{attribute 'OPC.UA.DA.StructuredType' := '1'}
FUNCTION_BLOCK FB_DosingPumpAgrowtek_R2_Batch EXTENDS FB_BaseDevice IMPLEMENTS I_PumpDosing

VAR_IN_OUT
	{attribute 'OPC.UA.DA' := '0'}
	//fbModbusMaster: FB_ModbusMaster;
	fbModbusManager: FB_ModbusManager;
	
	bInitialDose: BOOL := FALSE; // this is set to TRUE when the nDoseQTYMls is pre-loaded for the initial dose sequence. Setting nDoseQtyML or executing doses from control loops is disabled when this is true
END_VAR

VAR_INPUT
	nModbusUnitID: UINT; 
END_VAR

VAR
	// Modbus Variables
	nPumpID: UINT;	// Pump ID is different to the modbus ID because there are 5 pumps on the 1 modbus address
	 
	ePumpType: E_DosingPump;

	
	bEnableComms: BOOL := TRUE;
	bFirtRun: BOOL := TRUE;
	bResetTimer: BOOL := TRUE;
	
	// Async Statemachine Variables
	{attribute 'OPC.UA.DA' := '0'}
	eSMState: (WAIT, SET_TIME, GET_TIME, SET_SPEED, FINISH);
	
	// Dosing Variables
	{attribute 'OPC.UA.DA' := '0'} 
	fbTONdoseTime: TON;  
	{attribute 'OPC.UA.DA' := '1'} 
	nDoseRateMLph: UINT;
	{attribute 'OPC.UA.DA' := '1'} 
	nDoseQtyMls: REAL;
	{attribute 'OPC.UA.DA' := '1'} 
	tTimeToDose: TIME;
	
	nTimeToDoseSeconds: INT;
	nRetries: INT := 0;
	
	// delay between writing pump speed and reading pump speed
	fbTON_WaitForMsg : TON := (PT := T#1S);

	// Variables updated over Modbus
	{attribute 'OPC.UA.DA' := '1'} 
	nPumpSpeed_Requested: UINT;
	
	{attribute 'OPC.UA.DA' := '1'} 
	nPumpSpeed: UINT;
	{attribute 'OPC.UA.DA' := '1'} 
	nPumpRunTime: UINT; 
	
	
	
	
	bDoseRequestSent:		BOOL := FALSE;
	bDoseRequestComplete: 	BOOL := FALSE;
	
	tDataRefresh: TIME := T#10S;
	fbTON_DataRefresh: 	TON := (PT := tDataRefresh, IN := FALSE);
	fbTON_MsgTimeout: 	TON := (PT := T#4S, IN := FALSE);
	
	// Modbus Requests
	stModRead_MotorSpeed: 	ST_Modbus_ReadRequest;
	stModRead_MotorRunTime: ST_Modbus_ReadRequest;
	stModWrite_MotorSpeed: 	ST_Modbus_WriteRequest;
	stModWrite_SetID: 		ST_Modbus_WriteRequest;
	stModWrite_Timeout:	ST_Modbus_WriteRequest;
	stModRead_Timeout:	ST_Modbus_ReadRequest;
	
	
	bRaiseError1: BOOL := FALSE;
	bClearError: BOOL := FALSE;
	bRaiseError2: BOOL := FALSE;
	
	
END_VAR

fbTONdoseTime();
fbTON_MsgTimeout();
fbTON_DataRefresh();
fbTON_WaitForMsg();

IF GVL.bAutoUpdateDeviceState THEN
	eState := eStateTarget;	
END_IF

IF (eStateTarget = E_DeviceState.RUNNING) AND (eState := E_DeviceState.IDLE) THEN  // this is used to handle the initial batch dose commands from the sequene manager (this control loop uses the executeDOse method
	executeDose(DoseQtyMls := nDoseQtyMls, DoseRateMlph := 40, RequestComplete := ADR(bDoseRequestSent));
	eState := E_DeviceState.RUNNING;
END_IF


IF bFirtRun THEN
	init_ModbusRequests();
	bFirtRun := FALSE;
END_IF

IF eMode = E_DeviceMode.MANUAL THEN
	bEnable := TRUE;
END_IF


IF bResetTimer THEN
	fbTON_DataRefresh.IN := TRUE;
	bResetTimer := FALSE;
END_IF

// Asynchronous update of local variables from the Modbus request structures
nPumpSpeed 		:= WORD_TO_UINT(stModRead_MotorSpeed.ReadRegsVals[1]);
nPumpRunTime 	:= WORD_TO_UINT(stModRead_MotorRunTime.ReadRegsVals[1]);
	

CASE eSMState OF

	WAIT:
		eState := E_DeviceState.IDLE;
		fbTON_WaitForMsg(IN := FALSE);
		
	SET_TIME:
		eState := E_DeviceState.RUNNING;
		stModWrite_Timeout.WriteRegVals[1] := INT_TO_WORD(nTimeToDoseSeconds);
		fbModbusManager.addRequest_Write_Priority(WriteRequest := ADR(stModWrite_Timeout));
		fbTON_WaitForMsg(IN := TRUE);
		eSMState := GET_TIME;
		
		
	GET_TIME:
		IF stModRead_Timeout.ReadRegsVals[1] = INT_TO_WORD(nTimeToDoseSeconds) THEN
			stModRead_Timeout.ReadRegsVals[1] := 0;
			fbTON_WaitForMsg(IN := FALSE);
			eSMState := SET_SPEED;
		ELSE
			fbTON_WaitForMsg(IN := TRUE);
		END_IF
	
		IF fbTON_WaitForMsg.Q THEN
			fbModbusManager.addRequest_Read_Priority(ReadRequest := ADR(stModRead_Timeout));	
			fbTON_WaitForMsg(IN := FALSE);
		ELSE
			fbTON_WaitForMsg(IN := FALSE);			// add retry counter here
			nRetries := nRetries + 1;
			IF nRetries > 5 THEN
				eSMState := WAIT;
				eState := E_DeviceState.IDLE;
				bBusy := FALSE;
				nRetries := 0;
				raiseAlarm(Priority := E_AlarmPriority.High, Label := 'Motor Failed to Receive Duration Command After 5 Retries', Enabled := TRUE, DeviceAlarmID := 1);
			END_IF
		END_IF
		
	SET_SPEED:
		fbTON_WaitForMsg(IN := TRUE);
		
		IF fbTON_WaitForMsg.Q THEN
			stModWrite_MotorSpeed.WriteRegVals[1] := UINT_TO_WORD(nPumpSpeed_Requested);
			fbModbusManager.addRequest_Write_Priority(WriteRequest := stModWrite_MotorSpeed);
			fbTON_WaitForMsg(IN := FALSE);
			eSMState := FINISH;
		END_IF
		
	FINISH:
		fbTON_WaitForMsg(IN := TRUE);
		
		IF fbTON_WaitForMsg.Q THEN
			fbModbusManager.addRequest_Read_Priority(ReadRequest := ADR(stModRead_Timeout));	
			fbTON_WaitForMsg(IN := FALSE);
		END_IF
		
		IF stModRead_Timeout.ReadRegsVals[1] = 0 THEN
			eSMState := WAIT;
			bBusy := FALSE;
			eState := E_DeviceState.IDLE;
			bInitialDose := FALSE;
		ELSE
			nRetries := nRetries + 1;
			IF nRetries > 5 THEN
				raiseAlarm(Priority := E_AlarmPriority.High, Label := 'Motor Counter Failed to Reach 0 After 5 Retries', Enabled := TRUE, DeviceAlarmID := 2);
				nRetries := 0;
				bBusy := FALSE;
				eSMState := WAIT;
				eState := E_DeviceState.IDLE;
				bInitialDose := FALSE;	
			END_IF
		END_IF

END_CASE

{warning 'add method implementation '}
METHOD executeDose : BOOL
VAR_INPUT
	DoseQtyMls: LREAL;
	DoseRateMlph: UINT;
	RequestComplete: 	POINTER TO BOOL;
END_VAR
VAR_OUTPUT
	RequestAccepted: BOOL;
END_VAR
(* setDose dispenses the amount requested at a user requested dose rate *)

IF ((bEnable AND bEnableComms) OR (eMode = E_DeviceMode.MANUAL)) AND ( NOT bInitialDose)  THEN
	
		nPumpSpeed_Requested := 40;
		tTimeToDose := REAL_TO_TIME(( ABS(DoseQtyMls) / (480.0*(UINT_TO_REAL(nPumpSpeed_Requested)/100.0))) * 60.0 *1000.0);  // Agrowtek maximum flow rate is 480 ml/min
		fbTONdoseTime.PT := tTimeToDose;
	
		IF tTimeToDose >= T#1S THEN
			nTimeToDoseSeconds := (TIME_TO_INT(tTimeToDose)/1000);
			nDoseQtyMls := nTimeToDoseSeconds * ((nPumpSpeed_Requested/100.0) * (480.0/60.0));
			eSMState := SET_TIME;
			eState := E_Devicestate.RUNNING;
			bBusy := TRUE;	
		END_IF
	END_IF
END_METHOD

METHOD FB_init : BOOL


VAR_INPUT
	bInitRetains : BOOL; // if TRUE, the retain variables are initialized (warm start / cold start)
	bInCopyCode : BOOL;  // if TRUE, the instance afterwards gets moved into the copy code (online change)
	
	PumpID: STRING;
	PumpDescription: STRING;
	PumpType: E_DosingPump;
	ManifoldModbusID: UINT; 
	
END_VAR
sID := PumpID;
sDescr := PumpDescription;
ePumpType := PumpType;
nModbusUnitID := ManifoldModbusID;
END_METHOD

METHOD getAdrMotorTime : UINT
VAR_INPUT
	PumpType: E_DosingPump;
END_VAR
// This method retrieves the Modbus register for the individual Agrowtek pump
// We need to do this because 5 pumps share the same Modbus slave ID, however have differing registers to write to

CASE PumpType OF
	
	E_DosingPump.PH_DOWN:
		getAdrReadWriteSpeed := 200;
		
	E_DosingPump.NUTRIENT_A:
		getAdrReadWriteSpeed := 201;
		
	E_DosingPump.NUTRIENT_B:
		getAdrReadWriteSpeed := 202;
		
	E_DosingPump.NUTRIENT_C:
		getAdrReadWriteSpeed := 203;
		
	E_DosingPump.PH_UP:
		getAdrReadWriteSpeed := 204;
		
END_CASE
END_METHOD

METHOD getAdrReadAccumRunTime : UINT
VAR_INPUT
	PumpType: E_DosingPump;
END_VAR

VAR
	Address: UINT;
END_VAR
// This method retrieves the Modbus register for the individual Agrowtek pump
// We need to do this because 5 pumps share the same Modbus slave ID, however have differing registers to write to

CASE PumpType OF
	
	E_DosingPump.PH_DOWN:
		Address := 16#64;
		
	E_DosingPump.NUTRIENT_A:
		Address := 16#65;
		
	E_DosingPump.NUTRIENT_B:
		Address := 16#66;

	E_DosingPump.NUTRIENT_C:
		Address := 16#67;
		
	E_DosingPump.PH_UP:
		Address := 16#68;
		
END_CASE

getAdrReadAccumRunTime := Address;
END_METHOD

METHOD getAdrReadWriteSpeed : UINT
VAR_INPUT
	PumpType: E_DosingPump;
END_VAR
// This method retrieves the Modbus register for the individual Agrowtek pump
// We need to do this because 5 pumps share the same Modbus slave ID, however have differing registers to write to

CASE PumpType OF
	
	E_DosingPump.PH_DOWN:
		getAdrReadWriteSpeed := 16#64;
		
	E_DosingPump.NUTRIENT_A:
		getAdrReadWriteSpeed := 16#65;
		
	E_DosingPump.NUTRIENT_B:
		getAdrReadWriteSpeed := 16#66;
		
	E_DosingPump.NUTRIENT_C:
		getAdrReadWriteSpeed := 16#67;
		
	E_DosingPump.PH_UP:
		getAdrReadWriteSpeed := 16#68;
		
END_CASE
END_METHOD

METHOD init_ModbusRequests : BOOL
VAR_INPUT
END_VAR
stModRead_MotorSpeed.SlaveAddress := nModbusUnitID;			
stModRead_MotorSpeed.AdrFirstSlaveRegisterRead := getAdrReadWriteSpeed(PumpType := ePumpType);
stModRead_MotorSpeed.QtyWordsToRead := 1;				// The value is a 16-bit word
stModRead_MotorSpeed.bRequestAccepted := FALSE;
stModRead_MotorSpeed.bRequestCompleted := FALSE;
stModRead_MotorSpeed.ReadRegsVals := GVL.ModbusEmptyBuffer;

stModRead_MotorRunTime.SlaveAddress := nModbusUnitID;			
stModRead_MotorRunTime.AdrFirstSlaveRegisterRead := getAdrReadAccumRunTime(PumpType := ePumpType);
stModRead_MotorRunTime.QtyWordsToRead := 1;				// The value is a 32-bit word
stModRead_MotorRunTime.bRequestAccepted := FALSE;
stModRead_MotorRunTime.bRequestCompleted := FALSE;
stModRead_MotorRunTime.ReadRegsVals := GVL.ModbusEmptyBuffer;

stModWrite_Timeout.SlaveAddress := nModbusUnitID;
stModWrite_Timeout.AdrFirstSlaveRegisterWrite := getAdrMotorTime(PumpType := ePumpType);
stModWrite_Timeout.bRequestAccepted := FALSE;
stModWrite_Timeout.bRequestCompleted := FALSE;
stModWrite_Timeout.QtyWordsToWrite := 1;

stModRead_Timeout.SlaveAddress := nModbusUnitID;
stModRead_Timeout.AdrFirstSlaveRegisterRead := 200;
stModRead_Timeout.bRequestAccepted := FALSE;
stModRead_Timeout.bRequestCompleted := FALSE;
stModRead_Timeout.ReadRegsVals := GVL.ModbusEmptyBuffer;


stModWrite_MotorSpeed.SlaveAddress := nModbusUnitID;
stModWrite_MotorSpeed.AdrFirstSlaveRegisterWrite := getAdrMotorTime(PumpType := ePumpType);
stModWrite_MotorSpeed.bRequestAccepted := FALSE;
stModWrite_MotorSpeed.bRequestCompleted := FALSE;
stModWrite_MotorSpeed.QtyWordsToWrite := 1;

stModWrite_SetID.SlaveAddress := 254;
stModWrite_SetID.AdrFirstSlaveRegisterWrite := 0;
stModWrite_SetID.bRequestAccepted := FALSE;
stModWrite_SetID.bRequestCompleted := FALSE;
stModWrite_SetID.QtyWordsToWrite := 1;
END_METHOD

METHOD readSpeed : BOOL
VAR_INPUT
END_VAR
fbModbusManager.addRequest_Read_Priority(ReadRequest := ADR(stModRead_MotorSpeed));
END_METHOD

METHOD setDoseQTY_InitDose : BOOL
VAR_INPUT
	DoseQtyMls: INT;
END_VAR

nDoseQtyMls := DoseQtyMls;
bInitialDose := TRUE;
END_METHOD

METHOD setModID : BOOL
VAR_INPUT
	DesiredID: UINT;
END_VAR
stModWrite_SetID.WriteRegVals[1] := DesiredID;
fbModbusManager.addRequest_Write_Priority(WriteRequest := ADR(stModWrite_SetID));
END_METHOD

METHOD setOFF : BOOL
VAR_INPUT
	RequestComplete: 	POINTER TO BOOL;
END_VAR
VAR_OUTPUT
	RequestAccepted: 	BOOL;
END_VAR
eSMState := DOSING_OFF_TRIG;
END_METHOD

METHOD setON : BOOL
VAR_INPUT
	RateMlph	 : 		UINT;
	RequestComplete: 	POINTER TO BOOL;
END_VAR

VAR_OUTPUT
	RequestAccepted: 	BOOL;
END_VAR
END_METHOD

METHOD setSpeed99 : BOOL
VAR_INPUT
END_VAR
nPumpSpeed_Requested := 99;
stModWrite_MotorSpeed.WriteRegVals[1] := UINT_TO_WORD(nPumpSpeed_Requested);
fbModbusManager.addRequest_Write_Priority(WriteRequest := ADR(stModWrite_MotorSpeed));
END_METHOD

END_FUNCTION_BLOCK

(* stored: Version 1.1.0.1, ProductVersion 3.1.4024.12
   POU FB_DosingPumpAgrowtek_R2_Batch: Id {b6a0d439-38fc-4539-8bb5-7195aefa0850}, SpecialFunc None
   Method executeDose: Id {d340ae66-31b2-4241-98fd-adf67f20140e}
   Method FB_init: Id {af3d5559-23b2-4c09-9b37-5ccfffff8658}
   Method getAdrMotorTime: Id {04f191b6-822d-47fc-9ef0-c72cd17adcf8}
   Method getAdrReadAccumRunTime: Id {efda3fb4-a528-4d8d-b0de-b4e57ff04228}
   Method getAdrReadWriteSpeed: Id {871b1607-cc8d-464a-830f-d236f6b3d911}
   Method init_ModbusRequests: Id {f3f7a9a1-d1d0-4a9e-8c00-18e7ee927a95}
   Method readSpeed: Id {44ec65ec-c9f1-4087-b9e1-f5242d243cd2}
   Method setDoseQTY_InitDose: Id {7c559d95-b44d-4e4c-a647-8516394f035d}
   Method setModID: Id {86f67926-d322-4516-b147-b7737b226b50}
   Method setOFF: Id {3f1ba90b-7fab-4cd8-b5b7-2985e97f0df9}
   Method setON: Id {de8898c7-9e75-4b95-bb0d-efe23dd2d345}
   Method setSpeed99: Id {86fba625-9c18-43f7-80d0-9bcc1f95af53} *)
